FUNCTION_BLOCK Sequencer EXTENDS BaseConnector
VAR_INPUT
END_VAR
VAR_OUTPUT
END_VAR
VAR
	actions		: ARRAY[0..MAX_ACTION] OF StepAction;
	lastAction 	: INT := 0;
	currentAction : StepAction;
	startAction	: STRING;
	
	conditions	: ARRAY[0..99] OF StepCondition;
	lastCondition : INT := 0;
	currentCondition : StepCondition;
	
	timer		: TON;
	
END_VAR
VAR CONSTANT
	MAX_ACTION	: INT := 99;
END_VAR


timer(IN := TRUE, PT := MAX_TIME);

IF timer.ET > currentAction.timeout THEN
	
	ChangeStep(currentAction.timeoutAction);
ELSIF timer.ET > currentCondition.timeout THEN

	ChangeStep(currentCondition.timeoutAction);
END_IF

//IF currentConditon.satisfied THEN
	
//	ChangeStep(currentCondition.nextStep);
//END_IF

METHOD Bind : REFERENCE TO Transition
VAR_INPUT
	actionName	: STRING;
END_VAR
END_METHOD

METHOD ChangeStep : BOOL
VAR_INPUT
	actionName		: STRING;
END_VAR
VAR
	i : INT;
END_VAR
LogChange(currentAction.name, Condition, actionName);

FOR i := 0 TO MAX_ACTION DO
	IF (actions[i].name = actionName) THEN
		
		currentAction := actions[i];
	END_IF
END_FOR
END_METHOD

METHOD PRIVATE LogChange : BOOL
VAR_INPUT
	oldAction : STRING;
	satisfiedCondition : Condition;
	nextAction : STRING;
END_VAR
// TODO
END_METHOD

METHOD RegisterAction : BOOL
VAR_INPUT
	name			: STRING;
	caseNumber		: INT;
	timeout			: TIME;
	timeoutAction	: STRING;
	description		: STRING;
END_VAR
VAR
	a : REFERENCE TO StepAction REF= actions[lastAction];
END_VAR
a.name := name;
a.caseNumber := caseNumber;
a.timeout := timeout;
a.timeoutAction := timeoutAction;
a.description := description;

lastAction := lastAction + 1;
END_METHOD

METHOD RegisterCondition : REFERENCE TO Condition
VAR_INPUT
	name			: STRING;
	condition		: Condition;
	nextAction		: STRING;
	timeout			: TIME;
	timeoutAction	: STRING;
END_VAR
VAR
	c : REFERENCE TO StepCondition REF= conditions[lastAction];
END_VAR
c.name := name;
c.condition := condition;
c.nextAction := nextAction;
c.timeout := timeout;
c.timeoutAction := timeoutAction;

lastCondition := lastCondition + 1;
END_METHOD

METHOD Start : BOOL
VAR_INPUT
	startAction		: STRING;
END_VAR
this^.startAction := startAction; 

ChangeStep(startAction);
END_METHOD

END_FUNCTION_BLOCK

(* stored: Version 1.1.0.1, ProductVersion 3.1.4024.11
   POU Sequencer: Id {96f6bf52-4db2-4922-9ade-c20affde30d0}, SpecialFunc None
   Method Bind: Id {47e9fe29-6598-4e88-9005-0f5c4bb7df72}
   Method ChangeStep: Id {9cd436d0-78d3-48a5-89e7-03d922c3d837}
   Method LogChange: Id {4b28a56a-afbe-43ad-b2ae-8c249f80c93c}
   Method RegisterAction: Id {f8d51ba0-bd37-4d12-9644-bd208115b87e}
   Method RegisterCondition: Id {840e9851-9aaf-4dae-9629-426dcf8a91f9}
   Method Start: Id {5362ef16-7c50-4f2d-a7d6-f8f0db87a7bf} *)
